Staubli VAL3: get.pgx

public program get(string& x_sItem[] (dimensions=1), num x_nIndex (dimensions=1))
  local string l_sKey
  local num i
begin
  // start from the first
  l_sKey=first(saveProg:pProg)
  // search it
  while l_sKey!=""
    x_sItem=l_sKey
    l_sKey=next(saveProg:pProg[l_sKey])
    if i==x_nIndex
      return
    else
      i=i+1
    endIf
  endWhile
end
